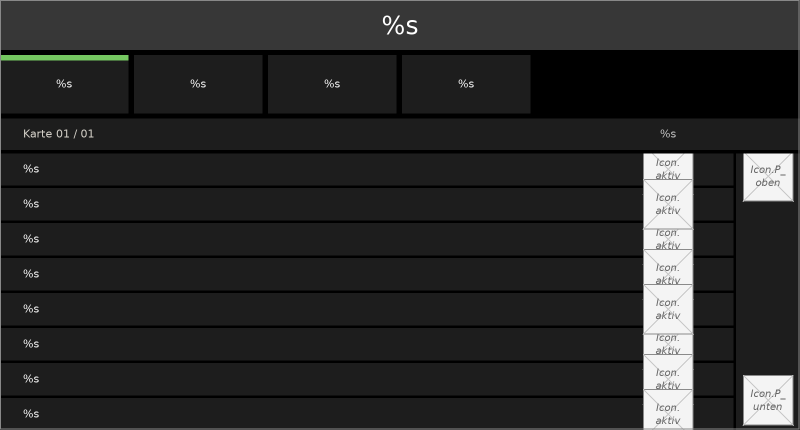
VISUALIZATION Liste_DI  // 800x430
VAR_IN_OUT

END_VAR
VAR
	i_verschieben:INT;


END_VAR
    Rectangle (736,153 64x277)
    Image (743,375 50x50), image: Icon.P_unten
        OnMouseClick: execute {
            IF i_verschieben<0 THEN
            	i_verschieben:=i_verschieben+35;
            End_if
        }
    Group (0,144 733x435)
        p2738717112: i_verschieben
        Rectangle (0,9 733x32)
        Rectangle (0,79 733x32)
        Rectangle (0,44 733x32)
        Rectangle (0,114 733x32)
        Rectangle (0,184 733x32)
        Rectangle (0,149 733x32)
        Rectangle (0,394 733x32)
        Rectangle (0,219 733x32)
        Rectangle (0,289 733x32)
        Rectangle (0,254 733x32)
        Rectangle (0,324 733x32)
        Rectangle (0,359 733x32)
        Rectangle (20,9 400x32), "%s"
        Image (643,0 50x50), image: Icon.inaktiv
        Image (643,0 50x50), image: Icon.aktiv
        Rectangle (20,79 400x32), "%s"
        Image (643,70 50x50), image: Icon.inaktiv
        Image (643,70 50x50), image: Icon.aktiv
        Rectangle (20,44 400x32), "%s"
        Image (643,35 50x50), image: Icon.inaktiv
        Image (643,35 50x50), image: Icon.aktiv
        Rectangle (20,114 400x32), "%s"
        Image (643,105 50x50), image: Icon.inaktiv
        Image (643,105 50x50), image: Icon.aktiv
        Rectangle (20,184 400x32), "%s"
        Image (643,175 50x50), image: Icon.inaktiv
        Image (643,175 50x50), image: Icon.aktiv
        Rectangle (20,149 400x32), "%s"
        Image (643,140 50x50), image: Icon.inaktiv
        Image (643,140 50x50), image: Icon.aktiv
        Rectangle (20,394 400x32), "%s"
        Image (643,385 50x50), image: Icon.inaktiv
        Image (643,385 50x50), image: Icon.aktiv
        Rectangle (20,219 400x32), "%s"
        Image (643,210 50x50), image: Icon.inaktiv
        Image (643,210 50x50), image: Icon.aktiv
        Rectangle (20,289 400x32), "%s"
        Image (643,280 50x50), image: Icon.inaktiv
        Image (643,280 50x50), image: Icon.aktiv
        Rectangle (20,254 400x32), "%s"
        Image (643,245 50x50), image: Icon.inaktiv
        Image (643,245 50x50), image: Icon.aktiv
        Rectangle (20,324 400x32), "%s"
        Image (643,315 50x50), image: Icon.inaktiv
        Image (643,315 50x50), image: Icon.aktiv
        Rectangle (20,359 400x32), "%s"
        Image (643,350 50x50), image: Icon.inaktiv
        Image (643,350 50x50), image: Icon.aktiv
    Image (743,151 50x50), image: Icon.P_oben
        OnMouseClick: execute {
            IF  i_verschieben>-100 THEN
            	i_verschieben:=i_verschieben-35;
            End_if
        }
    Group (0,118 800x32)
        Rectangle (0,0 800x32)
        Rectangle (20,0 324x32), "Karte 01 / 01"
        Rectangle (643,0 50x32), "%s", text list: 'Sprachen', text index: 49
    Rectangle (0,0 800x50), "%s", text list: 'Sprachen', text index: 44
    Rectangle (0,50 800x68)
    Rectangle (0,55 128x58), "%s", text list: 'Sprachen', text index: 45
        OnMouseClick: execute { GWP_Library.Visu.i_Frame_Index:=0; }
    Rectangle (134,55 128x58), "%s", text list: 'Sprachen', text index: 46
        OnMouseClick: execute { GWP_Library.Visu.i_Frame_Index:=1; }
    Rectangle (268,55 128x58), "%s", text list: 'Sprachen', text index: 47
        OnMouseClick: execute { GWP_Library.Visu.i_Frame_Index:=2; }
    Rectangle (402,55 128x58), "%s", text list: 'Sprachen', text index: 48
        OnMouseClick: execute { GWP_Library.Visu.i_Frame_Index:=3; }
    Rectangle (0,55 128x5)
    Rectangle (0,150 800x3)
END_VISUALIZATION

// VISUs/IBN/Liste_DO
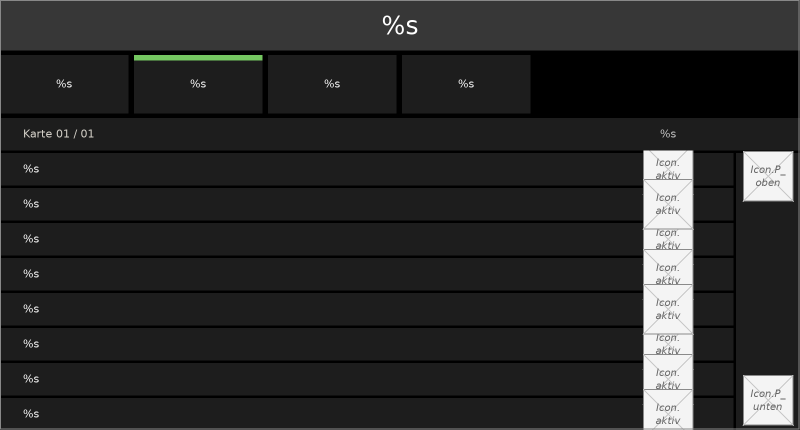
VISUALIZATION Liste_DO  // 800x430
    Rectangle (736,153 64x277)
    Image (743,375 50x50), image: Icon.P_unten
        OnMouseClick: execute {  }
    Image (743,151 50x50), image: Icon.P_oben
    Rectangle (0,153 733x32)
    Rectangle (0,223 733x32)
    Rectangle (0,188 733x32)
    Rectangle (0,258 733x32)
    Rectangle (0,328 733x32)
    Rectangle (0,293 733x32)
    Rectangle (0,538 733x32)
    Rectangle (0,363 733x32)
    Rectangle (0,433 733x32)
    Rectangle (0,398 733x32)
    Rectangle (0,468 733x32)
    Rectangle (0,503 733x32)
    Rectangle (20,153 400x32), "%s"
    Image (643,144 50x50), image: Icon.inaktiv
    Image (643,144 50x50), image: Icon.aktiv
    Rectangle (20,223 400x32), "%s"
    Image (643,214 50x50), image: Icon.inaktiv
    Image (643,214 50x50), image: Icon.aktiv
    Rectangle (20,188 400x32), "%s"
    Image (643,179 50x50), image: Icon.inaktiv
    Image (643,179 50x50), image: Icon.aktiv
    Rectangle (20,258 400x32), "%s"
    Image (643,249 50x50), image: Icon.inaktiv
    Image (643,249 50x50), image: Icon.aktiv
    Rectangle (20,328 400x32), "%s"
    Image (643,319 50x50), image: Icon.inaktiv
    Image (643,319 50x50), image: Icon.aktiv
    Rectangle (20,293 400x32), "%s"
    Image (643,284 50x50), image: Icon.inaktiv
    Image (643,284 50x50), image: Icon.aktiv
    Rectangle (20,538 400x32), "%s"
    Image (643,529 50x50), image: Icon.inaktiv
    Image (643,529 50x50), image: Icon.aktiv
    Rectangle (20,363 400x32), "%s"
    Image (643,354 50x50), image: Icon.inaktiv
    Image (643,354 50x50), image: Icon.aktiv
    Rectangle (20,433 400x32), "%s"
    Image (643,424 50x50), image: Icon.inaktiv
    Image (643,424 50x50), image: Icon.aktiv
    Rectangle (20,398 400x32), "%s"
    Image (643,389 50x50), image: Icon.inaktiv
    Image (643,389 50x50), image: Icon.aktiv
    Rectangle (20,468 400x32), "%s"
    Image (643,459 50x50), image: Icon.inaktiv
    Image (643,459 50x50), image: Icon.aktiv
    Rectangle (20,503 400x32), "%s"
    Image (643,494 50x50), image: Icon.inaktiv
    Image (643,494 50x50), image: Icon.aktiv
    Group (0,118 800x32)
        Rectangle (0,0 800x32)
        Rectangle (20,0 324x32), "Karte 01 / 01"
        Rectangle (643,0 50x32), "%s", text list: 'Sprachen', text index: 49
    Rectangle (0,0 800x50), "%s", text list: 'Sprachen', text index: 44
    Rectangle (0,55 128x58), "%s", text list: 'Sprachen', text index: 45
        OnMouseClick: execute { GWP_Library.Visu.i_Frame_Index:=0; }
    Rectangle (134,55 128x58), "%s", text list: 'Sprachen', text index: 46
        OnMouseClick: execute { GWP_Library.Visu.i_Frame_Index:=1; }
    Rectangle (268,55 128x58), "%s", text list: 'Sprachen', text index: 47
        OnMouseClick: execute { GWP_Library.Visu.i_Frame_Index:=2; }
    Rectangle (402,55 128x58), "%s", text list: 'Sprachen', text index: 48
        OnMouseClick: execute { GWP_Library.Visu.i_Frame_Index:=3; }
    Rectangle (0,55 128x5)
    Rectangle (134,55 128x5)
    Rectangle (268,55 128x5)
    Rectangle (402,55 128x5)
END_VISUALIZATION

// VISUs/IBN/SW_IBN_Einstellungen_K
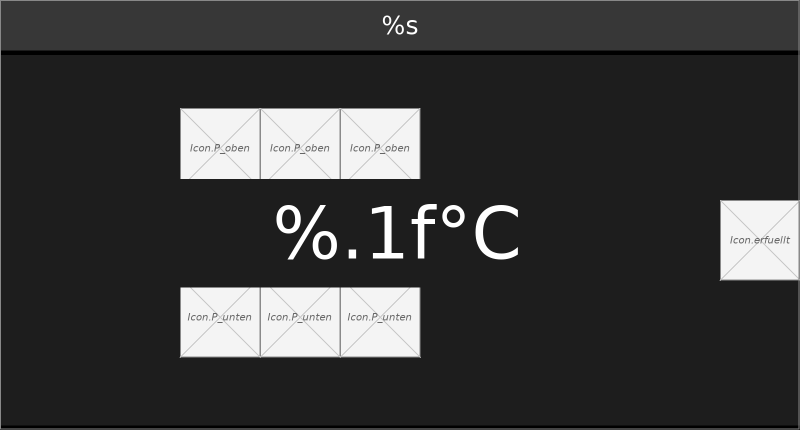
VISUALIZATION SW_IBN_Einstellungen_K  // 800x430
VAR_IN_OUT

END_VAR

VAR_INPUT
	i_titel:INT;
END_VAR
    Rectangle (0,0 800x50), "%s", text list: 'Sprachen', text index: i_titel
    Rectangle (0,55 800x370)
    Image (720,200 80x80), image: Icon.erfuellt
        OnMouseClick: execute { GWP_Library.Visu.i_Frame_Index:=0; }
    Image (180,108 80x80), image: Icon.P_oben
    Image (180,277 80x80), image: Icon.P_unten
    Image (260,108 80x80), image: Icon.P_oben
    Image (340,108 80x80), image: Icon.P_oben
        OnMouseClick: execute {  }
    Image (260,277 80x80), image: Icon.P_unten
    Image (340,277 80x80), image: Icon.P_unten
    Rectangle (110,179 415x108), "%.1f°C"
END_VISUALIZATION

// VISUs/Infoseite/Infoliste
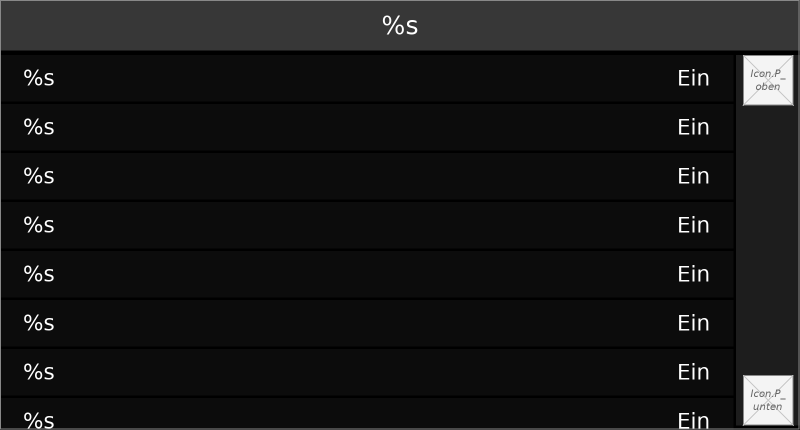
VISUALIZATION Infoliste  // 800x430
VAR_IN_OUT
	
END_VAR
VAR_INPUT
	i_Titel:INT;
	
END_VAR
VAR
	x_auf:BOOL;
	x_ab:BOOL;
	i_verschieben:INT:=0;
END_VAR
    Rectangle (0,0 800x50), "%s", text list: 'Sprachen', text index: i_Titel
    Rectangle (0,55 733x46)
    Label (20,55 479x46), "%s"
    Rectangle (0,104 733x46)
    Label (20,104 479x46), "%s"
    Rectangle (0,153 733x46)
    Label (20,153 479x46), "%s"
    Rectangle (0,202 733x46)
    Label (20,202 479x46), "%s"
    Rectangle (0,251 733x46)
    Label (20,251 479x46), "%s"
    Rectangle (0,300 733x46)
    Label (20,300 479x46), "%s"
    Rectangle (0,349 733x46)
    Label (20,349 479x46), "%s"
    Rectangle (583,55 130x46), "Ein"
    Rectangle (583,104 130x46), "Ein"
    Rectangle (0,398 733x46)
    Label (20,398 479x46), "%s"
    Rectangle (0,447 733x46)
    Label (20,447 479x46), "%s"
    Rectangle (0,496 733x46)
    Label (20,496 479x46), "%s"
    Rectangle (0,545 733x46)
    Label (20,545 479x46), "%s"
    Rectangle (583,545 130x46), "Ein"
    Rectangle (0,594 733x46)
    Label (20,594 479x46), "%s"
    Rectangle (583,153 130x46), "Ein"
    Rectangle (583,202 130x46), "Ein"
    Rectangle (583,251 130x46), "Ein"
    Rectangle (583,349 130x46), "Ein"
    Rectangle (583,300 130x46), "Ein"
    Rectangle (583,398 130x46), "Ein"
    Rectangle (583,447 130x46), "Ein"
    Rectangle (583,496 130x46), "Ein"
    Rectangle (583,594 130x46), "Ein"
    Group (736,55 64x370)
        Rectangle (0,0 64x370)
        Image (7,320 50x50), image: Icon.P_unten
            OnMouseClick:  ToggleVariable=x_ab
            OnMouseClick: execute {
                IF x_ab THEN
                	i_verschieben:=i_verschieben+50;
                	x_ab:=0;
                END_IF
            }
        Image (7,0 50x50), image: Icon.P_oben
            OnMouseClick:  ToggleVariable=x_auf
            OnMouseClick: execute {
                IF x_auf THEN
                	i_verschieben:=i_verschieben-50;
                	x_auf:=0;
                END_IF
            }
END_VISUALIZATION

// VISUs/Infoseite/Infoseite
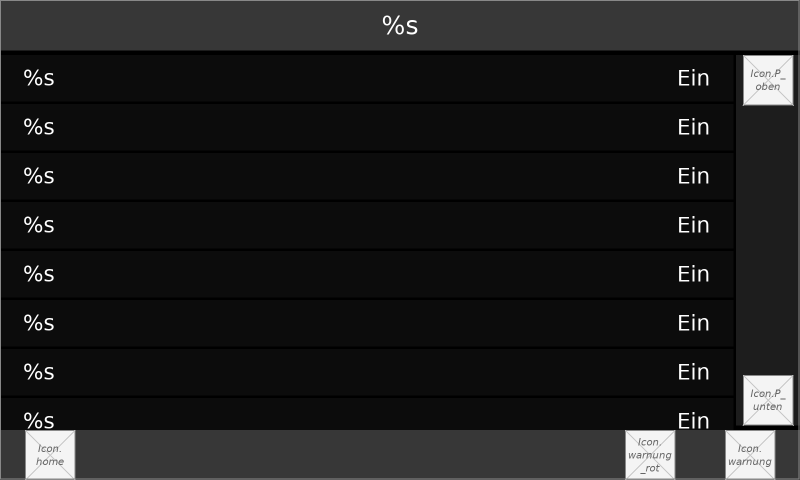
VISUALIZATION Infoseite  // 800x480
    Frame (0,0 800x430)
        shows Infoliste(i_Titel := 31)
    Frame (0,430 800x50)
        shows Fusszeile_50()
END_VISUALIZATION

// VISUs/Sollwertmenu_9/Sollwerte Einstellungen/SW_Einstellungen_C
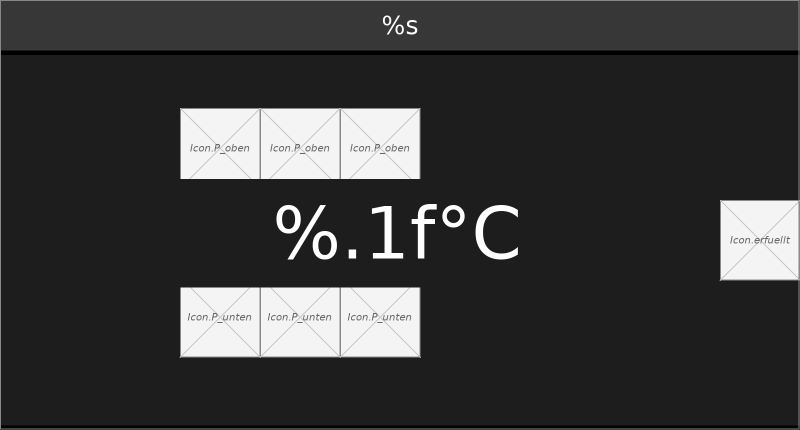
VISUALIZATION SW_Einstellungen_C  // 800x430
VAR_IN_OUT
		f_Data:REAL;
END_VAR

VAR_INPUT
	i_titel:INT;
END_VAR
    Rectangle (0,0 800x50), "%s", text list: 'Sprachen', text index: i_titel
    Rectangle (0,55 800x370), text variable: f_Data
    Image (720,200 80x80), image: Icon.erfuellt
        OnMouseClick: execute { GWP_Library.Visu.i_Frame_Index:=0; }
    Image (180,108 80x80), image: Icon.P_oben
        OnMouseClick: execute { f_Data:=f_Data +10; }
    Image (180,277 80x80), image: Icon.P_unten
        OnMouseClick: execute { f_Data:=f_Data -10; }
    Image (260,108 80x80), image: Icon.P_oben
        OnMouseClick: execute { f_Data:=f_Data +1; }
    Image (340,108 80x80), image: Icon.P_oben
        OnMouseClick: execute { f_Data:=f_Data +0.1; }
    Image (260,277 80x80), image: Icon.P_unten
        OnMouseClick: execute { f_Data:=f_Data -1; }
    Image (340,277 80x80), image: Icon.P_unten
        OnMouseClick: execute { f_Data:=f_Data -0.1; }
    Rectangle (110,179 415x108), "%.1f°C", text variable: f_Data
END_VISUALIZATION

// VISUs/Sollwertmenu_9/Sollwerte Einstellungen/SW_Einstellungen_Faktor
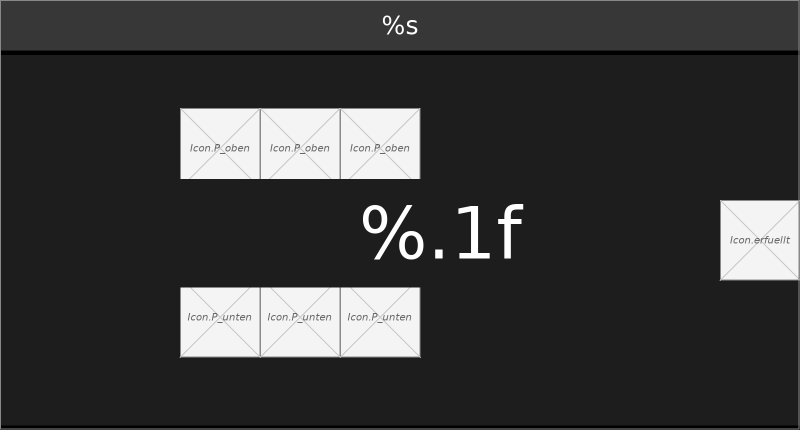
VISUALIZATION SW_Einstellungen_Faktor  // 800x430
VAR_IN_OUT
		f_Data:REAL;
END_VAR

VAR_INPUT
	i_titel:INT;
END_VAR
    Rectangle (0,0 800x50), "%s", text list: 'Sprachen', text index: i_titel
    Rectangle (0,55 800x370), text variable: f_Data
    Image (720,200 80x80), image: Icon.erfuellt
        OnMouseClick: execute { GWP_Library.Visu.i_Frame_Index:=0; }
    Image (180,108 80x80), image: Icon.P_oben
        OnMouseClick: execute { f_Data:=f_Data +10; }
    Image (180,277 80x80), image: Icon.P_unten
        OnMouseClick: execute { f_Data:=f_Data -10; }
    Image (260,108 80x80), image: Icon.P_oben
        OnMouseClick: execute { f_Data:=f_Data +1; }
    Image (340,108 80x80), image: Icon.P_oben
        OnMouseClick: execute { f_Data:=f_Data +0.1; }
    Image (260,277 80x80), image: Icon.P_unten
        OnMouseClick: execute { f_Data:=f_Data -1; }
    Image (340,277 80x80), image: Icon.P_unten
        OnMouseClick: execute { f_Data:=f_Data -0.1; }
    Rectangle (110,179 415x108), "%.1f", text variable: f_Data
END_VISUALIZATION

// VISUs/Sollwertmenu_9/Sollwerte Einstellungen/SW_Einstellungen_K
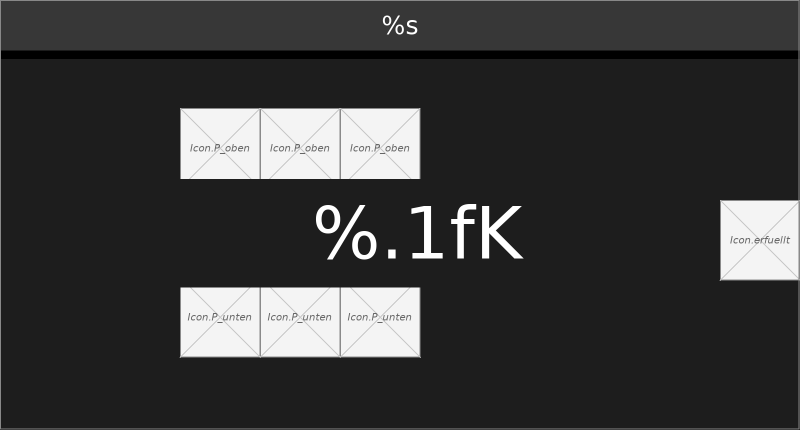
VISUALIZATION SW_Einstellungen_K  // 800x430
VAR_IN_OUT
		f_Data:REAL;
END_VAR

VAR_INPUT
	i_titel:INT;
END_VAR
    Rectangle (0,0 800x50), "%s", text list: 'Sprachen', text index: i_titel
    Rectangle (1,59 800x370), text variable: f_Data
    Image (720,200 80x80), image: Icon.erfuellt
        OnMouseClick: execute { GWP_Library.Visu.i_Frame_Index:=0; }
    Image (180,108 80x80), image: Icon.P_oben
        OnMouseClick: execute { f_Data:=f_Data +10; }
    Image (180,277 80x80), image: Icon.P_unten
        OnMouseClick: execute { f_Data:=f_Data -10; }
    Image (260,108 80x80), image: Icon.P_oben
        OnMouseClick: execute { f_Data:=f_Data +1; }
    Image (340,108 80x80), image: Icon.P_oben
        OnMouseClick: execute { f_Data:=f_Data +0.1; }
    Image (260,277 80x80), image: Icon.P_unten
        OnMouseClick: execute { f_Data:=f_Data -1; }
    Image (340,277 80x80), image: Icon.P_unten
        OnMouseClick: execute { f_Data:=f_Data -0.1; }
    Rectangle (110,179 415x108), "%.1fK", text variable: f_Data
END_VISUALIZATION

// VISUs/Sollwertmenu_9/Sollwerte Einstellungen/SW_Einstellungen_min
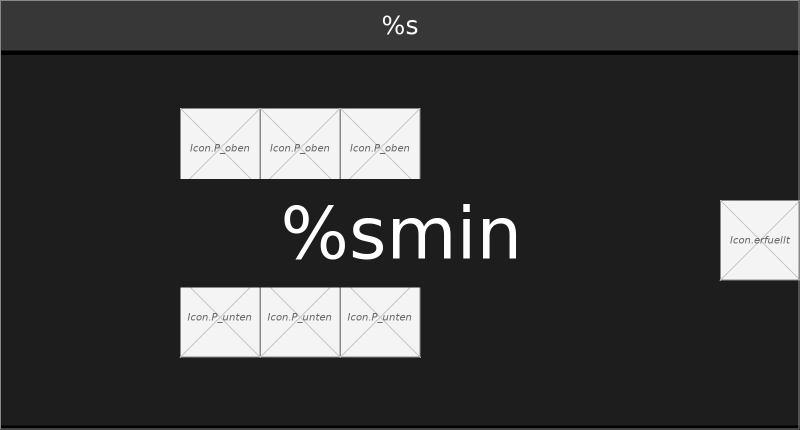
VISUALIZATION SW_Einstellungen_min  // 800x430
VAR_IN_OUT
		f_Data:WORD;
END_VAR

VAR_INPUT
	i_titel:INT;
END_VAR
    Rectangle (0,0 800x50), "%s", text list: 'Sprachen', text index: i_titel
    Rectangle (0,55 800x370), text variable: f_Data
    Image (720,200 80x80), image: Icon.erfuellt
        OnMouseClick: execute { GWP_Library.Visu.i_Frame_Index:=0; }
    Image (180,108 80x80), image: Icon.P_oben
        OnMouseClick: execute { f_Data:=f_Data +10; }
    Image (180,277 80x80), image: Icon.P_unten
        OnMouseClick: execute { f_Data:=f_Data -10; }
    Image (260,108 80x80), image: Icon.P_oben
        OnMouseClick: execute { f_Data:=f_Data +1; }
    Image (340,108 80x80), image: Icon.P_oben
        OnMouseClick: execute { f_Data:=f_Data +0.1; }
    Image (260,277 80x80), image: Icon.P_unten
        OnMouseClick: execute { f_Data:=f_Data -1; }
    Image (340,277 80x80), image: Icon.P_unten
        OnMouseClick: execute { f_Data:=f_Data -0.1; }
    Rectangle (110,179 415x108), "%smin", text variable: f_Data
END_VISUALIZATION

// VISUs/Sollwertmenu_9/Sollwerte Einstellungen/SW_Einstellungen_ms
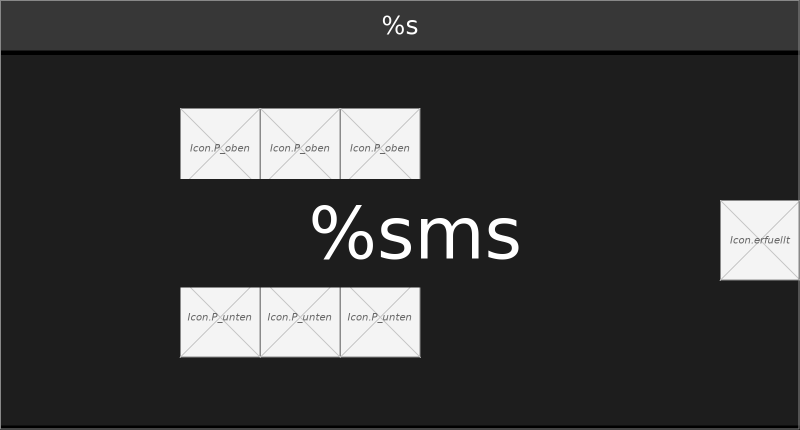
VISUALIZATION SW_Einstellungen_ms  // 800x430
VAR_IN_OUT
		f_Data:WORD;
END_VAR

VAR_INPUT
	i_titel:INT;
END_VAR
    Rectangle (0,0 800x50), "%s", text list: 'Sprachen', text index: i_titel
    Rectangle (0,55 800x370), text variable: f_Data
    Image (720,200 80x80), image: Icon.erfuellt
        OnMouseClick: execute { GWP_Library.Visu.i_Frame_Index:=0; }
    Image (180,108 80x80), image: Icon.P_oben
        OnMouseClick: execute { f_Data:=f_Data +10; }
    Image (180,277 80x80), image: Icon.P_unten
        OnMouseClick: execute { f_Data:=f_Data -10; }
    Image (260,108 80x80), image: Icon.P_oben
        OnMouseClick: execute { f_Data:=f_Data +1; }
    Image (340,108 80x80), image: Icon.P_oben
        OnMouseClick: execute { f_Data:=f_Data +0.1; }
    Image (260,277 80x80), image: Icon.P_unten
        OnMouseClick: execute { f_Data:=f_Data -1; }
    Image (340,277 80x80), image: Icon.P_unten
        OnMouseClick: execute { f_Data:=f_Data -0.1; }
    Rectangle (110,179 415x108), "%sms", text variable: f_Data
END_VISUALIZATION

// VISUs/Sollwertmenu_9/Sollwerte Einstellungen/SW_zuruecksetzen
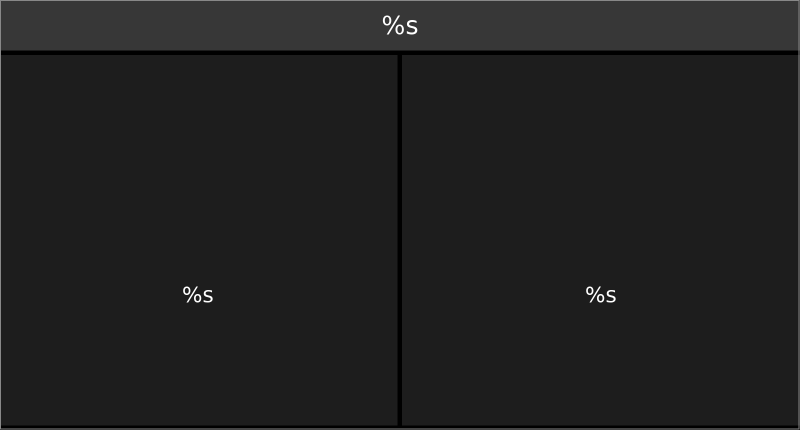
VISUALIZATION SW_zuruecksetzen  // 800x430
VAR_IN_OUT
	x_Zuruecksetzen:BOOL;
END_VAR

VAR_OUTPUT
	

END_VAR

VAR_INPUT
	i_Titel:INT;
	i_Text_1:INT;
	i_Text_2:INT;	

	
END_VAR
    Rectangle (0,0 800x50), "%s", text list: 'Sprachen', text index: i_Titel
    Rectangle (0,55 397x370)
        OnMouseClick: execute { GWP_Library.Visu.i_Frame_Index:=0; }
    Rectangle (0,55 397x5)
    Rectangle (123,280 150x30), "%s", text list: 'Sprachen', text index: i_Text_1
    Polygon (943,131)
    Rectangle (402,55 398x370)
        OnMouseDown: execute { x_Zuruecksetzen:=TRUE; }
        OnMouseUp: execute { x_Zuruecksetzen:=false; }
    Rectangle (402,55 398x5)
    Rectangle (402,280 398x30), "%s", text list: 'Sprachen', text index: i_Text_2
END_VISUALIZATION

// VISUs/Sollwertmenu_9/Sollwertmenu/Sollwertmenu
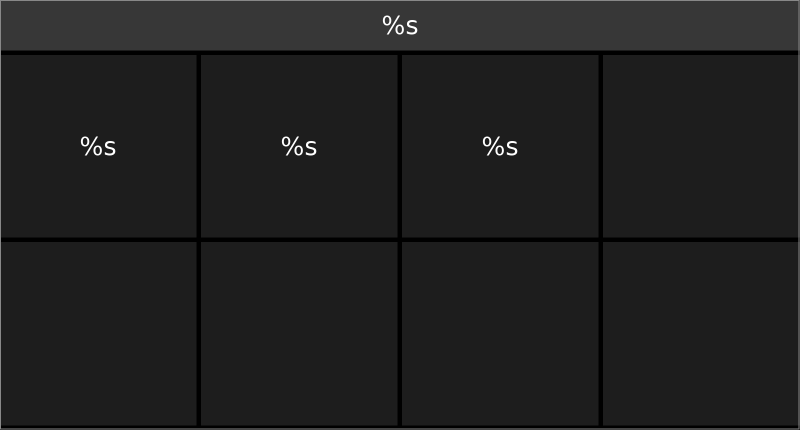
VISUALIZATION Sollwertmenu  // 800x430
    Rectangle (0,0 800x50), "%s", text list: 'Sprachen', text index: 3
    Rectangle (0,55 196x182), "%s", text list: 'Sprachen', text index: 0
        OnMouseClick:  Assign=Sollwertmenu_Waermegewinnung, Type=Assignment
    Rectangle (201,55 196x182), "%s", text list: 'Sprachen', text index: 1
        OnMouseClick:  Assign=Sollwertmenu_Waermepumpe, Type=Assignment
    Rectangle (402,55 196x182), "%s", text list: 'Sprachen', text index: 2
        OnMouseClick:  Assign=Sollwertmenu_Waermesenke, Type=Assignment
    Rectangle (603,55 197x182)
    Rectangle (0,242 196x183)
    Rectangle (201,242 196x183)
    Rectangle (402,242 196x183)
    Rectangle (603,242 197x183)
    Frame (0,430 800x50)
        shows Fusszeile_50()
    Image (125,430 50x50), image: Icon.zurueck
        OnMouseClick:  Assign=Hauptmenu, Type=Assignment
END_VISUALIZATION

// VISUs/Sollwertmenu_9/Wärmegewinnung/UWP/SW_WG_UWP_Verd
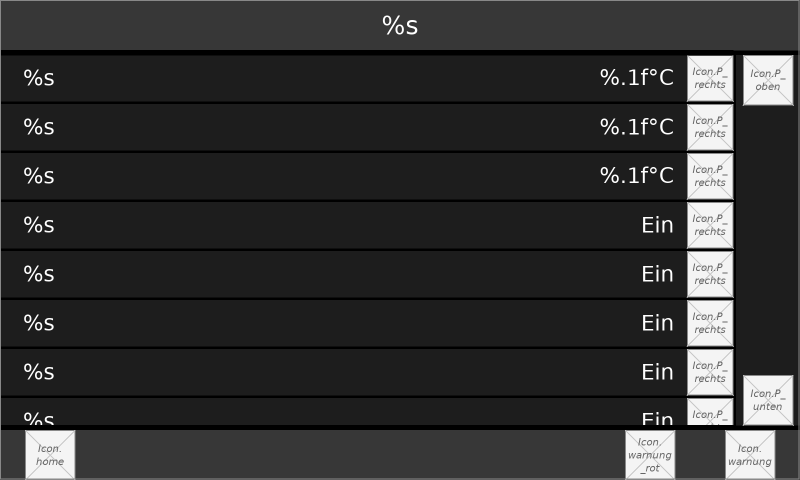
VISUALIZATION SW_WG_UWP_Verd  // 800x480
VAR_IN_OUT
	FB_GR2:GR_2;
END_VAR
    Frame (0,0 800x430), frame switch variable: GWP_Library.Visu.i_Frame_Index
        shows SW_WG_UWP_Verd_Liste(i_Titel := 25, FB_GR2 := FB_GR2)
        shows SW_Einstellungen_Zeit(i_titel := 53, f_Data := FB_GR2.f_AT)
        shows SW_Einstellungen_C(i_titel := 30, f_Data := FB_GR2.f_RefPunkt_TO1)
        shows SW_Einstellungen_C_1(i_titel := 31, f_Data := FB_GR2.f_SW_Min)
        shows SW_Einstellungen_Zeit(i_titel := 30)
    Frame (0,430 800x50)
        shows Fusszeile_50()
END_VISUALIZATION

// VISUs/Sollwertmenu_9/Wärmegewinnung/UWP/SW_WG_UWP_Verd_Liste
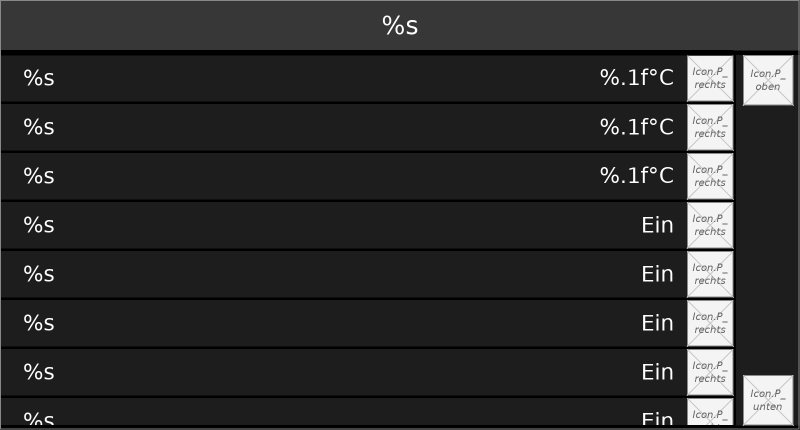
VISUALIZATION SW_WG_UWP_Verd_Liste  // 800x430
VAR_IN_OUT
	FB_GR2:GR_2;
END_VAR

VAR_INPUT
	i_Titel:INT;
END_VAR

VAR
	i_verschieben:INT;
 END_VAR
    Rectangle (0,55 733x46)
    Label (20,55 479x46), "%s"
    Rectangle (0,104 733x46)
    Label (20,104 479x46), "%s"
    Rectangle (547,55 130x45), "%.1f°C", text variable: FB_GR2.f_AT
    Rectangle (547,104 130x46), "%.1f°C", text variable: FB_GR2.f_RefPunkt_TO1
    Image (687,55 46x46), image: Icon.P_rechts
        OnMouseClick: execute { GWP_Library.Visu.i_Frame_Index:=1; }
    Image (687,104 46x46), image: Icon.P_rechts
        OnMouseClick: execute { GWP_Library.Visu.i_Frame_Index:=2; }
    Rectangle (0,153 733x46)
    Label (20,153 479x46), "%s"
    Rectangle (0,202 733x46)
    Label (20,202 479x46), "%s"
    Rectangle (0,251 733x46)
    Label (20,251 479x46), "%s"
    Rectangle (0,300 733x46)
    Label (20,300 479x46), "%s"
    Rectangle (0,349 733x46)
    Label (20,349 479x46), "%s"
    Rectangle (0,398 733x46)
    Label (20,398 479x46), "%s"
    Rectangle (0,447 733x46)
    Label (20,447 479x46), "%s"
    Rectangle (0,496 733x46)
    Label (20,496 479x46), "%s"
    Rectangle (0,545 733x46)
    Label (20,545 479x46), "%s"
    Rectangle (547,153 130x45), "%.1f°C", text variable: FB_GR2.f_SW_Min
        OnMouseClick: execute { GWP_Library.Visu.i_Frame_Index:=2; }
    Rectangle (547,202 130x46), "Ein"
    Rectangle (547,251 130x46), "Ein"
    Rectangle (547,300 130x46), "Ein"
    Rectangle (547,349 130x46), "Ein"
    Rectangle (547,447 130x46), "Ein"
    Rectangle (547,398 130x46), "Ein"
    Rectangle (547,496 130x46), "Ein"
    Rectangle (547,545 130x46), "Ein"
    Image (687,153 46x46), image: Icon.P_rechts
        OnMouseClick: execute { GWP_Library.Visu.i_Frame_Index:=3; }
    Image (687,545 46x46), image: Icon.P_rechts
    Image (687,496 46x46), image: Icon.P_rechts
    Image (687,447 46x46), image: Icon.P_rechts
    Image (687,398 46x46), image: Icon.P_rechts
    Image (687,349 46x46), image: Icon.P_rechts
    Image (687,300 46x46), image: Icon.P_rechts
    Image (687,251 46x46), image: Icon.P_rechts
    Image (687,202 46x46), image: Icon.P_rechts
    Rectangle (0,594 733x46)
    Label (20,594 479x46), "%s"
    Rectangle (547,594 130x45), "Ein"
    Image (687,594 46x46), image: Icon.P_rechts
    Image (79,430 50x50), image: Icon.zurueck
        OnMouseClick:  Assign=Sollwertmenu_Waermegewinnung, Type=Assignment
        OnMouseClick: execute { i_verschieben:=0; }
    Rectangle (0,0 800x50), "%s", text list: 'Sprachen', text index: i_Titel
    Group (736,55 64x370)
        Rectangle (0,0 64x370)
        Image (7,320 50x50), image: Icon.P_unten
            OnMouseClick: execute {
                IF i_verschieben<0 THEN
                	i_verschieben:=i_verschieben+53;
                End_if
            }
        Image (7,0 50x50), image: Icon.P_oben
            OnMouseClick: execute {
                IF  i_verschieben>-200 THEN
                	i_verschieben:=i_verschieben-53;
                End_if
            }
    Rectangle (0,50 733x5)
    Rectangle (0,425 733x5)
END_VISUALIZATION

// VISUs/Sollwertmenu_9/Wärmegewinnung/Kachel_Abtauspeicher
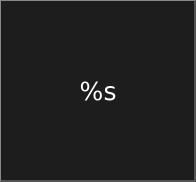
VISUALIZATION Kachel_Abtauspeicher  // 196x182
    Rectangle (0,0 196x182), "%s", text list: 'Sprachen', text index: 10
END_VISUALIZATION

// VISUs/Sollwertmenu_9/Wärmegewinnung/Kachel_Abtauungen
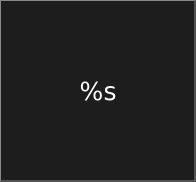
VISUALIZATION Kachel_Abtauungen  // 196x182
    Rectangle (0,0 196x182), "%s", text list: 'Sprachen', text index: 11
END_VISUALIZATION

// VISUs/Sollwertmenu_9/Wärmegewinnung/Kachel_Abwaerme
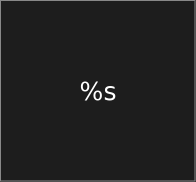
VISUALIZATION Kachel_Abwaerme  // 196x182
    Rectangle (0,0 196x182), "%s", text list: 'Sprachen', text index: 12
END_VISUALIZATION

// VISUs/Sollwertmenu_9/Wärmegewinnung/Kachel_Erdsonden
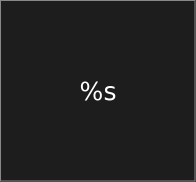
VISUALIZATION Kachel_Erdsonden  // 196x182
    Rectangle (0,0 196x182), "%s", text list: 'Sprachen', text index: 6
END_VISUALIZATION

// VISUs/Sollwertmenu_9/Wärmegewinnung/Kachel_Grundwasser
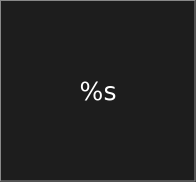
VISUALIZATION Kachel_Grundwasser  // 196x182
    Rectangle (0,0 196x182), "%s", text list: 'Sprachen', text index: 7
END_VISUALIZATION

// VISUs/Sollwertmenu_9/Wärmegewinnung/Kachel_Luft
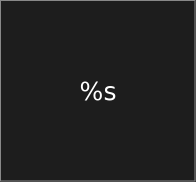
VISUALIZATION Kachel_Luft  // 196x182
    Rectangle (0,0 196x182), "%s", text list: 'Sprachen', text index: 8
END_VISUALIZATION

// VISUs/Sollwertmenu_9/Wärmegewinnung/Kachel_Tiefhaltung
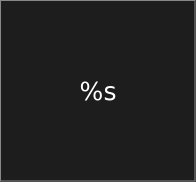
VISUALIZATION Kachel_Tiefhaltung  // 196x182
    Rectangle (0,0 196x182), "%s", text list: 'Sprachen', text index: 9
END_VISUALIZATION

// VISUs/Sollwertmenu_9/Wärmegewinnung/Kachel_UWP_Verd
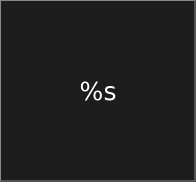
VISUALIZATION Kachel_UWP_Verd  // 196x182
    Rectangle (0,0 196x182), "%s", text list: 'Sprachen', text index: 5
END_VISUALIZATION

// VISUs/Sollwertmenu_9/Wärmegewinnung/Sollwertmenu_Waermegewinnung
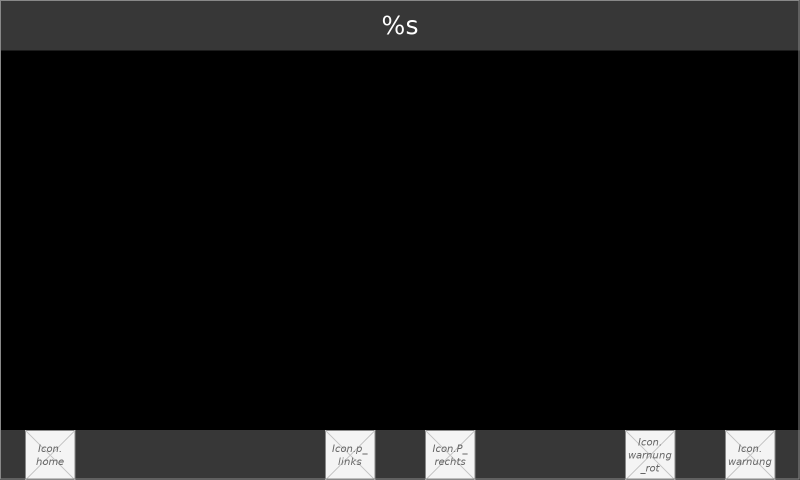
VISUALIZATION Sollwertmenu_Waermegewinnung  // 800x480
VAR_IN_OUT
		
END_VAR

VAR
	i_verschieben:INT;

END_VAR
    Image (425,430 50x50), image: Icon.reinnavigieren
    Image (325,430 50x50), image: Icon.reinnavigieren
    Rectangle (0,0 800x50), "%s", text list: 'Sprachen', text index: 4
    Frame (0,430 800x50)
        shows Fusszeile_50()
    Image (425,430 50x50), image: Icon.P_rechts
        OnMouseClick: execute {
            IF i_verschieben>-800 THEN
            	i_verschieben:=i_verschieben-800;
            END_IF
        }
    Image (325,430 50x50), image: Icon.p_links
        OnMouseClick: execute {
            IF i_verschieben<0 THEN
            	i_verschieben:=i_verschieben+800;
            END_IF
        }
    Rectangle (88,515 454x57), "Kachel 1: 0;55 *** Kachel 2: 201;55 *** Kachel 3: 402;55 *** Kachel 4: 604;55 Kachel 5: 0;242 *** Kachel 6: 201;242 *** Kachel 7: 402;242 *** Kachel 8: 604;242"
END_VISUALIZATION

// VISUs/Sollwertmenu_9/Wärmepumpe/EEV/SW_WP_EEV
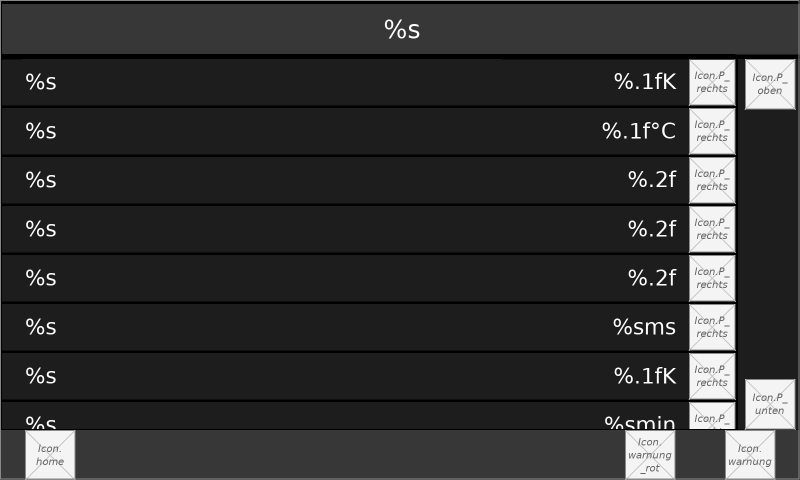
VISUALIZATION SW_WP_EEV  // 800x480
VAR_IN_OUT
	FB_EEV:EEV;
	
END_VAR
	
VAR_INPUT
	

END_VAR
    Frame (2,4 800x430), frame switch variable: GWP_Library.Visu.i_Frame_Index
        shows SW_WP_EEV_Liste(i_Titel := i_verschieben, FB_EEV := FB_EEV)
        shows SW_Einstellungen_K(i_titel := 30, f_Data := FB_EEV.f_SollwertUBH)
        shows SW_Einstellungen_C(i_titel := 30, f_Data := FB_EEV.f_MOP)
        shows SW_Einstellungen_Faktor(i_titel := 30, f_Data := FB_EEV.f_PFaktor)
        shows SW_Einstellungen_Faktor(i_titel := 30, f_Data := FB_EEV.f_IFaktor)
        shows SW_Einstellungen_Faktor(i_titel := 30, f_Data := FB_EEV.f_DFaktor)
        shows SW_Einstellungen_ms(i_titel := 30, f_Data := FB_EEV.t_Takt.wMilliseconds)
        shows SW_Einstellungen_K(i_titel := 30, f_Data := FB_EEV.f_MinUBH)
        shows SW_Einstellungen_min(i_titel := 30, f_Data := FB_EEV.t_AL_EEV.wMinute)
        shows SW_zuruecksetzen(i_Titel := 72, i_Text_1 := 73, i_Text_2 := 72, x_Zuruecksetzen := FB_EEV.x_SW_Reset)
    Frame (0,430 800x50)
        shows Fusszeile_50()
END_VISUALIZATION

// VISUs/Sollwertmenu_9/Wärmepumpe/EEV/SW_WP_EEV_Liste
